% RSLogix 500 project part 1.RSS, saved by version 8.40.00.08 %
PROJECT "UNTITLED"    % processor: MicroLogix 1400 %

PROGRAM FILES
  LAD 2   2 rungs

DATA FILES
  O0 OUTPUT  6 elements
  I1 INPUT  8 elements
  S2 STATUS  66 elements
  B3 BINARY  1 elements
  T4 TIMER  1 elements
  C5 COUNTER  1 elements
  R6 CONTROL  1 elements
  N7 INTEGER  1 elements
  F8 FLOAT  1 elements

LADDER 2
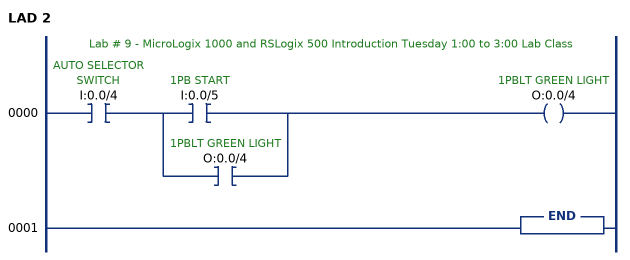
% Rung: 0 %  % edit flag set %
% Lab # 9 - MicroLogix 1000 and RSLogix 500 Introduction Tuesday 1:00 to 3:00 Lab Class %
SOR XIC I:0.0/4 BST XIC I:0.0/5 NXB XIC O:0.0/4 BND OTE O:0.0/4 EOR
%   I:0.0/4  "AUTO SELECTOR SWITCH" %
%   I:0.0/5  "1PB START" %
%   O:0.0/4  "1PBLT GREEN LIGHT" %
% Rung: 1 %
SOR END EOR
